Fanuc TP program (LS listing): INIT.LS

/PROG  INIT
/ATTR
OWNER		= MNEDITOR;
COMMENT		= "";
PROG_SIZE	= 163;
CREATE		= DATE 25-06-05  TIME 09:24:20;
MODIFIED	= DATE 25-06-05  TIME 09:24:20;
FILE_NAME	= ;
VERSION		= 0;
LINE_COUNT	= 0;
MEMORY_SIZE	= 407;
PROTECT		= READ_WRITE;
TCD:  STACK_SIZE	= 0,
      TASK_PRIORITY	= 50,
      TIME_SLICE	= 0,
      BUSY_LAMP_OFF	= 0,
      ABORT_REQUEST	= 0,
      PAUSE_REQUEST	= 0;
DEFAULT_GROUP	= 1,*,*,*,*;
CONTROL_CODE	= 00000000 00000000;
LOCAL_REGISTERS	= 0,0,0;
/APPL

AUTO_SINGULARITY_HEADER;
  ENABLE_SINGULARITY_AVOIDANCE   : TRUE;
/MN
/POS
/END
